FUNCTION_BLOCK FB_TwinExtruder EXTENDS FB_GCodeTool IMPLEMENTS I_Dispenser
VAR
	pFbHeaterRef	: POINTER TO FB_MZHeaterRef;
	pFirstExtruder 	: POINTER TO FB_Extruder;
	pSecondExtruder	: POINTER TO FB_Extruder;
	///****************************************Aktionvariablen****************************************************
	
	//Action: "Extrude"
	bExtrude			: BOOL;
	nStateA_Extrude		: USINT;
	nExtrudeDistance	: DINT;
	nExtrudeCtrl		: DINT;
	
	nCurrentTemp		: UINT;
END_VAR
VAR CONSTANT
	cNumberOfSlots: UINT := 4; //Slot für Exposure hinzugefügt
END_VAR

SUPER^();	//FB_MzTool aufrufen

IF bExtrude THEN	//Extrudieren
	A_Extrude();
	IF nStateA_Extrude >= 80 THEN
		IF nStateA_Extrude >= 99 THEN
			bError := TRUE;
		END_IF
		bExtrude := FALSE;
		nStateA_Extrude := 0;
		M_RemoveListEntry(nSearchValue:= E_Action.ACTION_Extrude);
	END_IF
END_IF

//Prozessdaten aktualisieren
IF pFbHeaterRef > 0 THEN
	stProcessData.n32Data[7] := BOOL_TO_DINT(pFbHeaterRef^.bHeaterIsOn);
	nCurrentTemp := pFbHeaterRef^.nTemp3Actual;
	stProcessData.n32Data[8] := nCurrentTemp;
END_IF

IF pFirstExtruder > 0 AND pSecondExtruder > 0 THEN
	stProcessData.n32Data[9] := BOOL_TO_DINT(pFirstExtruder^.P_bIsExtruding OR pSecondExtruder^.P_bIsExtruding);
END_IF

aObjProcData[nNotifyId] := stProcessData;

ACTION A_Extrude:
IF pFirstExtruder^.P_bError THEN
	stError.ErrorId := pFirstExtruder^.P_nErrorId;
	stError.POUState := nStateA_Extrude;
	nStateA_Extrude := 99;
END_IF

IF nStateA_Extrude <> 99 THEN
	IF pSecondExtruder^.P_bError THEN
		stError.ErrorId := pSecondExtruder^.P_nErrorId;
		stError.POUState := nStateA_Extrude;
		nStateA_Extrude := 99;
	END_IF	
END_IF

CASE nStateA_Extrude OF
	0:	MEMSET(ADR(stActionData),0,SIZEOF(stActionData));
		stActionData.eAction := E_Action.ACTION_Extrude;
		stActionData.aParams[1] := nExtrudeDistance; 
		stActionData.aParams[2] := nExtrudeCtrl;
		stError.ErrorId := pFirstExtruder^.M_ExeAction(stActionData);
		IF stError.ErrorId = 0 THEN
			stError.ErrorId := pSecondExtruder^.M_ExeAction(stActionData);
			IF stError.ErrorId = 0 THEN
				nStateA_Extrude := 1;
			ELSE //FirstExtruder wieder stoppen
				nStateA_Extrude := 99;
			END_IF
		ELSE
			nStateA_Extrude := 99;
		END_IF
		
	1:	//ready ?
		IF NOT(pFirstExtruder^.M_GetActionBusy(E_Action.ACTION_Extrude) OR 
				pSecondExtruder^.M_GetActionBusy(E_Action.ACTION_Extrude)) THEN
			nStateA_Extrude := 80;
		END_IF
		
	70:	//Stoppen
		pFirstExtruder^.M_CancelAction(E_Action.ACTION_Extrude);
		pSecondExtruder^.M_CancelAction(E_Action.ACTION_Extrude);
		nStateA_Extrude := 71;
		
	71:	IF NOT(pFirstExtruder^.M_GetActionBusy(E_Action.ACTION_Extrude) OR 
			pSecondExtruder^.M_GetActionBusy(E_Action.ACTION_Extrude)) THEN
			nStateA_Extrude := 80;
		END_IF
END_CASE

IF nStateA_Extrude = 99 THEN
	pFirstExtruder^.M_CancelAction(E_Action.ACTION_Extrude);
	pSecondExtruder^.M_CancelAction(E_Action.ACTION_Extrude);
	stError.Cmd := E_Action.ACTION_Extrude;
	stError.POU := E_POU.POU_FB_TwinExtruder;
	stError.POUAction := E_POUACT.POUACT_A_Extrude;
	fbErrorList.M_Add(stError);	
END_IF
END_ACTION

ACTION A_Reset:
nStateA_ResetSpec := 80;
SUPER^.A_Reset();
END_ACTION

ACTION A_Stop:
IF nStateA_Stop = 0 THEN

	nStateA_Stop := 1;
END_IF

SUPER^.A_Stop();
END_ACTION

METHOD FB_init : BOOL
VAR_INPUT
	bInitRetains : BOOL; // if TRUE, the retain variables are initialized (warm start / cold start)
	bInCopyCode : BOOL;  // if TRUE, the instance afterwards gets moved into the copy code (online change)
END_VAR
eObjectType := E_ObjectType.OBJECTTYPE_TwinExtruder;
eObjectGroup := E_ObjectGroup.OBJECTGROUP_MzTool OR E_ObjectGroup.OBJECTGROUP_Device;
END_METHOD

METHOD M_AddChild : ERRORID
VAR_INPUT
	pObject : POINTER TO FB_Object;
	nSlotNr	: UINT;
	nIndex 	: INT;
END_VAR
//Kann folgende Objekt-Typen aufnehmen
//Extruder, Nozzle, Exposure
IF pObject > 0 THEN
	IF pObject^.P_eObjectType = E_ObjectType.OBJECTTYPE_Extruder OR
		pObject^.P_eObjectType = E_ObjectType.OBJECTTYPE_DummyTool OR
		pObject^.P_eObjectType = E_ObjectType.OBJECTTYPE_Exposure OR
		pObject^.P_eObjectType = E_ObjectType.OBJECTTYPE_Nozzle THEN
		M_AddChild := SUPER^.M_AddChild(pObject,nSlotNr,nIndex);
	ELSE
		M_AddChild := E_ErrorIdObjMgmt.ERRORID_InvalidParentObject;
	END_IF
ELSE
	M_AddChild := E_ErrorIdObjMgmt.ERRORID_InvalidParentObject;
END_IF
END_METHOD

METHOD M_CancelAction
VAR_INPUT
	eAction : E_Action;
END_VAR
IF eAction = E_Action.ACTION_Extrude THEN
	IF bExtrude AND nStateA_Extrude < 70 THEN
		nStateA_Extrude := 70;
	END_IF
ELSE
	SUPER^.M_CancelAction(eAction);
END_IF
END_METHOD

METHOD M_CheckAction : ERRORID
VAR_INPUT
	refActionData	: REFERENCE TO ST_ActionData;
	pCorrelObject	: POINTER TO FB_Object;
END_VAR
CASE refActionData.eAction OF
	E_Action.ACTION_Extrude, //BasicAction für ActionOnArray
	E_Action.ACTION_CleanTip,
	E_Action.ACTION_MeasureTool,
	E_Action.ACTION_TeachTarget:
		RETURN;
ELSE
	M_CheckAction := SUPER^.M_CheckAction(refActionData, pCorrelObject);
END_CASE
END_METHOD

METHOD M_CheckProcDataType : BOOL
VAR_INPUT
	eProcDataType : E_ProcDataType;
END_VAR
IF eProcDataType = E_ProcDataType.PROCDATATYPE_Temp1 THEN
	M_CheckProcDataType := TRUE;
END_IF
END_METHOD

METHOD M_CheckProps : ERRORID
VAR_INPUT
END_VAR

VAR
	pSlot : POINTER TO FB_Slot;
END_VAR
M_CheckProps := SUPER^.M_CheckProps();
//TwinExtruder muss zwingend zwei Childs als Extruder besitzen
//auf Slot1 -> FirstExtruder
//auf Slot2 -> SecondExtruder
pFirstExtruder := 0;
pSecondExtruder := 0;

pSlot := fbSlotList.M_GetAtNr(1);
IF pSlot > 0 THEN
	IF pSlot^.P_pChild > 0 THEN
		IF pSlot^.P_pChild^.P_eObjectType = E_ObjectType.OBJECTTYPE_Extruder THEN
			pFirstExtruder := pSlot^.P_pChild;
		END_IF
	END_IF
END_IF

pSlot := fbSlotList.M_GetAtNr(2);
IF pSlot > 0 THEN
	IF pSlot^.P_pChild > 0 THEN
		IF pSlot^.P_pChild^.P_eObjectType = E_ObjectType.OBJECTTYPE_Extruder THEN
			pSecondExtruder := pSlot^.P_pChild;
		END_IF
	END_IF
END_IF

IF pFirstExtruder = 0 OR pSecondExtruder = 0 THEN
	M_CheckProps := E_ErrorIdObjMgmt.ERRORID_UnusedExtruderSlot;
END_IF

IF pPiece = 0 THEN
	M_CheckProps := E_ErrorIdObjMgmt.ERRORID_NoNozzleOnTool;
END_IF
END_METHOD

METHOD M_DispenserPrepare : ERRORID
VAR_INPUT
END_VAR
END_METHOD

METHOD M_DispenserStart : ERRORID
VAR_INPUT
END_VAR

VAR
	stActionData : ST_ActionData;
END_VAR
stActionData.eAction := E_ACTION.ACTION_Extrude;
stActionData.aParams[2] := 1;
M_DispenserStart := M_ExeAction(stActionData);
END_METHOD

METHOD M_DispenserStop : ERRORID
VAR_INPUT
END_VAR

VAR
	stActionData : ST_ActionData;
END_VAR
stActionData.eAction := E_ACTION.ACTION_Extrude;
M_DispenserStop := M_ExeAction(stActionData);
END_METHOD

METHOD M_ExeAction : ERRORID
VAR_INPUT
	refActionData : REFERENCE TO ST_ActionData;	
END_VAR
IF NOT (eCurrentState = E_MachineState.MACHINESTATE_Idle OR
	eCurrentState = E_MachineState.MACHINESTATE_Active OR
	eCurrentState = E_MachineState.MACHINESTATE_Ready) THEN
	M_ExeAction := E_ErrorIdCmd.ERRORID_InvalidState;
	RETURN;
END_IF

CASE refActionData.eAction OF
		E_Action.ACTION_Extrude:
			//Beide Extruder gelockt?
			IF NOT (pFirstExtruder^.P_bIsLocked AND pSecondExtruder^.P_bIsLocked) THEN
				M_ExeAction := E_ErrorIdCmd.ERRORID_DeviceNotLocked;
				RETURN;				
			END_IF
			
			nExtrudeDistance := refActionData.aParams[1]; 
			nExtrudeCtrl := refActionData.aParams[2];
			
			IF NOT bExtrude AND nExtrudeCtrl = 1 THEN //Einschalten
				bExtrude := TRUE;
				fbList.A_AddHeadValue(hList := hList, putValue := E_Action.ACTION_Extrude);
			ELSIF bExtrude AND nExtrudeCtrl = 0 THEN //Ausschalten
				MEMSET(ADR(stActionData),0,SIZEOF(stActionData));
				stActionData.eAction := E_Action.ACTION_Extrude;
				stActionData.aParams[1] := nExtrudeDistance; 
				stActionData.aParams[2] := nExtrudeCtrl := 0; 
				pFirstExtruder^.M_ExeAction(stActionData);
				pSecondExtruder^.M_ExeAction(stActionData);
			ELSE
				RETURN;
			END_IF
			
	ELSE
		M_ExeAction := SUPER^.M_ExeAction(refActionData);
		RETURN;
END_CASE

bBusy := TRUE;
eCurrentState := E_MachineState.MACHINESTATE_Active;
END_METHOD

METHOD M_GetAllProps : ERRORID
VAR_INPUT
	refCmdData : REFERENCE TO  ST_CmdData;
END_VAR

VAR
	i : UINT;
	pToolSlot	: POINTER TO FB_Slot;
END_VAR
//BaseProperties lesen
SUPER^.M_GetAllProps(refCmdData);

nCurrentPropIndex := nCurrentPropIndex + 1;
IF pFbHeaterRef > 0 THEN
	refCmdData.n32Data[nCurrentPropIndex] := 1;	
END_IF
END_METHOD

METHOD M_GetProcData : DINT
VAR_INPUT
	eProcDataType : E_ProcDataType;
END_VAR
IF eProcDataType = E_ProcDataType.PROCDATATYPE_Temp1 THEN
	M_GetProcData := nCurrentTemp;
END_IF
END_METHOD

METHOD M_SetAllProps : ERRORID
VAR_INPUT
	refCmdData : REFERENCE TO  ST_CmdData;
END_VAR

VAR
	nParentMzToolObjId	: UINT;
	pParentTool 		: POINTER TO FB_MzTool;
	pParentHead 		: POINTER TO FB_MzHead;
END_VAR
M_SetAllProps := SUPER^.M_SetAllProps(refCmdData);

IF M_SetAllProps > 0 THEN
	RETURN;
END_IF

//Spezi-Paramter schreiben
nCurrentPropIndex := nCurrentPropIndex + 1;
nSpecPropIndex := nCurrentPropIndex;

IF refCmdData.n32Data[nCurrentPropIndex] = 1 THEN
	pFbHeaterRef := ADR(pFbMultiZ^.aFbHeaterRef[7]);
ELSE
	pFbHeaterRef := 0;
END_IF

nNoOfProps := nCurrentPropIndex + 1;
END_METHOD

METHOD M_SetPrintParams : ST_MethResult
VAR_INPUT
	eType 		: E_PrintParamType;
	nNumerator	: USINT;
	nValue		: DINT;
END_VAR

VAR
	stActionData : ST_ActionData;
END_VAR
IF eType = E_PrintParamType.Feed THEN
	IF nNumerator = 1 THEN
		IF pFirstExtruder > 0 THEN
			M_SetPrintParams.nErrorId := pFirstExtruder^.M_SetFeed(DINT_TO_UINT(nValue));	
		END_IF	
	ELSIF nNumerator = 2 THEN
		IF pSecondExtruder > 0 THEN
			M_SetPrintParams.nErrorId := pSecondExtruder^.M_SetFeed(DINT_TO_UINT(nValue));	
		END_IF	
	ELSE
		M_SetPrintParams.nErrorId := E_ErrorIdCmd.ERRORID_InvalidPrintParamNumerator;
	END_IF
ELSE
	M_SetPrintParams.nErrorId := E_ErrorIdCmd.ERRORID_InvalidPrintParamType;
END_IF

IF M_SetPrintParams.nErrorId > 0 THEN
	M_SetPrintParams.bError := TRUE;
END_IF
END_METHOD

PROPERTY P_bSensorMounted : BOOL
GET
P_bSensorMounted:= pFirstExtruder^.P_bSensorMounted OR pSecondExtruder^.P_bSensorMounted;
END_GET
END_PROPERTY

PROPERTY P_eDispenserState : E_DispenserState
GET
IF pFirstExtruder > 0 AND_THEN pFirstExtruder^.P_bIsExtruding THEN
	P_eDispenserState := E_DispenserState.Dispensing;
END_IF

IF pSecondExtruder > 0 AND_THEN pSecondExtruder^.P_bIsExtruding THEN
	P_eDispenserState := E_DispenserState.Dispensing;
END_IF
END_GET
END_PROPERTY

PROPERTY P_pFirstExtruder : POINTER TO FB_Extruder
GET
P_pFirstExtruder := pFirstExtruder;
END_GET
END_PROPERTY

PROPERTY P_pSecondExtruder : POINTER TO FB_Extruder
GET
P_pSecondExtruder := pSecondExtruder;
END_GET
END_PROPERTY

END_FUNCTION_BLOCK

(* stored: Version 1.1.0.1, ProductVersion 3.1.4024.9
   POU FB_TwinExtruder: Id {300af7ef-d10a-480b-b935-d39fdb3a4c95}, SpecialFunc None
   Action A_Extrude: Id {1246c239-7047-421a-a83e-a0666c614861}
   Action A_Reset: Id {ff7b46b0-98cf-4617-98ce-ed260c20d10b}
   Action A_Stop: Id {3aeb04dc-21fb-4fc7-a5d7-52fd59033583}
   Method FB_init: Id {d3c5cb36-6527-4621-885b-df1928cb9d14}
   Method M_AddChild: Id {3c1e8d65-84d3-4441-bf9b-33b30da1b41c}
   Method M_CancelAction: Id {96a40542-11aa-4280-a016-195724e6cb6d}
   Method M_CheckAction: Id {bc514dc4-4725-42b0-b8ee-b3d6a89863d8}
   Method M_CheckProcDataType: Id {fd295005-4c82-4b39-a70c-a2984e92f9ca}
   Method M_CheckProps: Id {97e5631f-b319-4d49-bfd7-49976179b76b}
   Method M_DispenserPrepare: Id {5e5c0125-3449-47e8-82aa-e10ebee34902}
   Method M_DispenserStart: Id {5633c960-0ecb-4d8d-99c4-07fda63d317a}
   Method M_DispenserStop: Id {2e7f500c-4ad5-4929-bb29-1ac8ba016c21}
   Method M_ExeAction: Id {07745b7b-a7f9-409d-80b6-804834e62aae}
   Method M_GetAllProps: Id {c4cfc590-1c5d-4425-99f4-65f114c35961}
   Method M_GetProcData: Id {3e859ee6-01a3-424b-8c8e-f9dfd14f4ff1}
   Method M_SetAllProps: Id {27d7e9a9-f223-4985-b808-da155916ea7c}
   Method M_SetPrintParams: Id {6a71f872-c97d-4742-afc7-db499fe68c28}
   Property P_bSensorMounted: Id {7f851516-e469-472b-9094-9da8664e4e9c}
   Get Get: Id {47688e52-0486-4486-9650-bb6762603ef3}
   Property P_eDispenserState: Id {41ac99da-c9b4-4be3-a146-6c51e8b5ea5b}
   Get Get: Id {d0646265-c163-44ab-869c-b102d8d5253c}
   Property P_pFirstExtruder: Id {36ec6037-7550-4176-a53c-28ebd74e826e}
   Get Get: Id {1bb52ad6-8ad7-4e29-a142-f33b69ebdc01}
   Property P_pSecondExtruder: Id {23b1cd7c-6a53-48af-88d3-fb06bd77d5cd}
   Get Get: Id {e0c73aeb-6bd9-4576-9661-e309b4e00bee} *)
